# EPICS substitutions: vactrlApp/Db/sr-ut-temperature.substitutions
file sr-ut-temperature.template
{
	pattern { INDX	}
		{ 1	}
		{ 2	}
		{ 3 	}
		{ 4	}
		{ 5	}
}
